FUNCTION_BLOCK Motor
VAR_INPUT
	nMotorNum :DINT ;
END_VAR
VAR_OUTPUT
	nMotorValue : DINT;
END_VAR
VAR
	nMotorSpin : DINT;
END_VAR

nMotorSpin := nMotorSpin + 1;

END_FUNCTION_BLOCK

(* stored: Version 1.1.0.1, ProductVersion 3.1.4024.16
   POU Motor: Id {7892ad7d-03d2-41b4-ab0b-76862df00861}, SpecialFunc None *)
